// TIA Portal V19 export
FUNCTION "@CmMotor" : Void   // FC2004, STL
TITLE = Control Module for Motor/Pump - Fixed Speed
{ S7_Optimized_Access := 'FALSE' }
AUTHOR : FoodSystem(AlfaLaval)
FAMILY : ControlModule
NAME : CM005
VERSION : 3.5
// Date        Rev      Change                                           Changed by
// ---------------------------------------------------------------------------------------------------------------------------------
// 08.04.2022 V3.0       Update                                    Food System (Alfalaval)
// 
// 28.07.2022 V3.1       Update                                    Food System (Alfalaval)
// 
// 14.11.2022 V3.2       Update                                    Food System (Alfalaval)
// 
// 26.12.2022 V3.3       Update                                    Food System (Alfalaval)
// 
// 16.05.2023 V3.4       Update                                    Food System (Alfalaval)
// 
// 01.12.2023 V3.5       Update                                    Food System (Alfalaval)
// ---------------------------------------------------------------------------------------------------------------------------------
// Motor with 3 Inputs and 1 output
// 1. Running Feedback, 2. Tripped Feedback, 3. Remote Feedback
// and 1. Start O/P
// The CM_Motor controls and monitors a single-speed one direction motor. 
// Additionally it also supports functions like feedback monitoring and alarm 
// generation, simulation and displays status to the HMI
// Date        Rev      Change                                           Changed by
// ---------------------------------------------------------------------------------------------------------------------------------
// 08.04.2022 V3.0       Update                                    Food System (Alfalaval)
// 
// 28.07.2022 V3.1       Update                                    Food System (Alfalaval)
// 
// 14.11.2022 V3.2       Update                                    Food System (Alfalaval)
// ---------------------------------------------------------------------------------------------------------------------------------
// Motor with 3 Inputs and 1 output
// 1. Running Feedback, 2. Tripped Feedback, 3. Remote Feedback
// and 1. Start O/P
// The CM_Motor controls and monitors a single-speed one direction motor. 
// Additionally it also supports functions like feedback monitoring and alarm 
// generation, simulation and displays status to the HMI
// stored: AutoNumber false
   VAR_INPUT
      i_Remote : Bool;   // Local / Remote
      i_RunFb : Bool;   // Motor Run Feedback
      i_TrippedFb : Bool;   // Motor Tripped Feedback
      i_Inhibit : Bool;   // 0 = Interlock, 1 = Healthy. Motor Inhibit
      i_EStop : Bool;   // Emergency Stop
      FeatureITripPolarity : Bool;   // Set 0 (I_TrippedFb --> 0 = Tripped), Set 1 (I_TrippedFb --> 1 = Tripped) Only for Trip HW Signal.
      FirstScanBit : Bool;   // First Scan Bit
      OneSec : Bool;   // One Second Pulse
      SimOn : Bool;   // Activate Simulation
      SimOff : Bool;   // Deactivate Simulation
      CommonReset : Bool;   // Reset fault
      HooterReset : Bool;   // Reset Hooter
      AutoReqMode : Bool;   // Activate PLC Auto Mode
      DCSOperation : Bool;   // Request from DCS to operate command from DCS
   END_VAR
   VAR_OUTPUT
      q_On : Bool;   // Motor run output
   END_VAR
   VAR_IN_OUT
      CM : Any;   // Parameter for control module
   END_VAR
   VAR_TEMP
      UDTMotor : "UDT CM_Motor";   // UDT data for for control module
      Pointer : DWord;   // Pointer for storage UDT
      DB : Word;   // UDT DB for data load
      TempQAutoOn : Bool;   // Internal on command in Auto mode before start interlock
      TempQManON : Bool;   // Internal on command in manual mode
      Permissive : Struct   // Temp Bits for Start Interlock Processing
         Inlk0 : Bool;
         Inlk1 : Bool;
         Inlk2 : Bool;
         Inlk3 : Bool;
         Inlk4 : Bool;
         Inlk5 : Bool;
         Inlk6 : Bool;
         Inlk7 : Bool;
         Inlk8 : Bool;
         Inlk9 : Bool;
         Inlk10 : Bool;
         Inlk11 : Bool;
         Inlk12 : Bool;
         Inlk13 : Bool;
         Inlk14 : Bool;
         Inlk15 : Bool;
      END_STRUCT;
      Interlock : Struct   // Temp Bits for Run Interlock Processing
         Inlk0 : Bool;
         Inlk1 : Bool;
         Inlk2 : Bool;
         Inlk3 : Bool;
         Inlk4 : Bool;
         Inlk5 : Bool;
         Inlk6 : Bool;
         Inlk7 : Bool;
         Inlk8 : Bool;
         Inlk9 : Bool;
         Inlk10 : Bool;
         Inlk11 : Bool;
         Inlk12 : Bool;
         Inlk13 : Bool;
         Inlk14 : Bool;
         Inlk15 : Bool;
      END_STRUCT;
      BypassPermissive : Struct   // Temp Bits for Bypass Start Interlock Processing
         Inlk0 : Bool;
         Inlk1 : Bool;
         Inlk2 : Bool;
         Inlk3 : Bool;
         Inlk4 : Bool;
         Inlk5 : Bool;
         Inlk6 : Bool;
         Inlk7 : Bool;
         Inlk8 : Bool;
         Inlk9 : Bool;
         Inlk10 : Bool;
         Inlk11 : Bool;
         Inlk12 : Bool;
         Inlk13 : Bool;
         Inlk14 : Bool;
         Inlk15 : Bool;
      END_STRUCT;
      BypassInterlock : Struct   // Temp Bits for Bypass Run Interlock Processing
         Inlk0 : Bool;
         Inlk1 : Bool;
         Inlk2 : Bool;
         Inlk3 : Bool;
         Inlk4 : Bool;
         Inlk5 : Bool;
         Inlk6 : Bool;
         Inlk7 : Bool;
         Inlk8 : Bool;
         Inlk9 : Bool;
         Inlk10 : Bool;
         Inlk11 : Bool;
         Inlk12 : Bool;
         Inlk13 : Bool;
         Inlk14 : Bool;
         Inlk15 : Bool;
      END_STRUCT;
   END_VAR
BEGIN

NETWORK
TITLE = LOAD DATA FROM DB

      L     P##CM;  // Any datapointer for CM
      LAR1;
      L     W [AR1, P#4.0];
      T     #DB;  // Number of DB
      L     D [AR1, P#6.0];
      T     #Pointer;  // Pointer for data
      LAR1;

      OPN   DB [#DB];
      L     W [AR1, P#0.0];  // Data transfer to Local Area
      T     %LW0;

      L     W [AR1, P#2.0];  // Data transfer to Local Area
      T     %LW2;


      L     W [AR1, P#4.0];  // Data transfer to Local Area
      T     %LW4;

      L     W [AR1, P#6.0];  // Data transfer to Local Area
      T     %LW6;


      L     W [AR1, P#8.0];  // Data transfer to Local Area
      T     #UDTMotor.FTRSet;

      L     W [AR1, P#10.0];  // Data transfer to Local Area
      T     #UDTMotor.FTSSet;

      L     W [AR1, P#12.0];  // Data transfer to Local Area
      T     #UDTMotor.FTRActual;

      L     W [AR1, P#14.0];  // Data transfer to Local Area
      T     #UDTMotor.FTSActual;

      L     W [AR1, P#16.0];  // Data transfer to Local Area
      T     #UDTMotor.ARH;

      L     W [AR1, P#18.0];  // Data transfer to Local Area
      T     #UDTMotor.Display;

      L     W [AR1, P#20.0];  // Data transfer to Local Area
      T     #UDTMotor.TempARH;


      L     W [AR1, P#22.0];  // Data transfer to Local Area
      T     #UDTMotor.PulseTimeStart;

      L     W [AR1, P#24.0];  // Data transfer to Local Area
      T     #UDTMotor.PulseTimeStop;

      L     W [AR1, P#26.0];  // Data transfer to Local Area
      T     #UDTMotor.BypassPermissive;

      L     W [AR1, P#28.0];  // Data transfer to Local Area
      T     #UDTMotor.BypassInterlock;

      L     W [AR1, P#30.0];  // Data transfer to Local Area
      T     %LW30;

      L     W [AR1, P#32.0];  // Data transfer to Local Area
      T     %LW32;

      L     W [AR1, P#34.0];  // Data transfer to Local Area
      T     #UDTMotor.AlarmHmi;

      L     W [AR1, P#36.0];  // Data transfer to Local Area
      T     #UDTMotor.ActiveTime;


      L     W [AR1, P#38.0];  // Data transfer to Local Area
      T     #UDTMotor.MotorType;

      L     D [AR1, P#40.0];  // Data transfer to Local Area
      T     #UDTMotor.Spare2;

      L     D [AR1, P#44.0];  // Data transfer to Local Area
      T     %LD44;  // oBJECT enable

      L     W [AR1, P#48.0];  // Data transfer to Local Area
      T     %LW48;  // FP EDGES


NETWORK
TITLE = RESET MANUAL COMMAND AND RESET ALARMS BY FIRST_SCAN_BIT
// On Power on and Off Motor start commond should reset.
      A     #FirstScanBit;  // First Scan
      R     #UDTMotor.Command.ManRun;  // Manual Start Commonad
      R     #UDTMotor.Status.FTR;  // Motor/Pump Fail to Run Fault.(FTR)
      R     #UDTMotor.Status.FTS;  // Motor/Pump Fail to Stop Fault.(FTS)


NETWORK
TITLE = Operation from DCS=1 (Disable command buttons from HMI)
      A     #DCSOperation;
      ON    #i_Remote;
      =     #UDTMotor.Command.DCSOperation;
      =     #UDTMotor.ObjEn.AlarmMask;
      =     #UDTMotor.ObjEn.Auto;
      =     #UDTMotor.ObjEn.Manual;
      =     #UDTMotor.ObjEn.ByInlk;
      =     #UDTMotor.ObjEn.ByPer;
      =     #UDTMotor.ObjEn.FTRSetpointEn;
      =     #UDTMotor.ObjEn.FTSSetpointEn;
      =     #UDTMotor.ObjEn.Reset;
      =     #UDTMotor.ObjEn.SimOn;
      =     #UDTMotor.ObjEn.ResetARH;

      A     #DCSOperation;
      ON    #i_Remote;
      O     #UDTMotor.Status.Mode;
      =     #UDTMotor.ObjEn.Start;


NETWORK
TITLE = LOAD INTERLOCK TO TEMP
// ----------------------------------------------------------------------------------------------//
//                                  READ INTERLOCK STATUS TO TEMP                                 //
// ----------------------------------------------------------------------------------------------//
      L     %LW30;  // Load start intrlocks
      T     %LW62;  // Save into TEMP
      L     %LW32;  // Load run intrlocks
      T     %LW64;  // Save into TEMP
      L     #UDTMotor.BypassPermissive;  // Load bypass start intrlocks
      T     %LW66;  // Save into TEMP
      L     #UDTMotor.BypassInterlock;  // Load bypass run intrlocks
      T     %LW68;  // Save into TEMP


NETWORK
TITLE = Reset Start Permissive & Run Interlock Bypasses
      A     #UDTMotor.Command.ResetRunPermissiveILByp;  // Check if Reset Interlock Bypass Bit is True

      JCN   INTBYPS_RST;  // Jump if the Reset Interlock Bypass bit is False

      L     16#0;
      T     #UDTMotor.BypassInterlock;  // Transfer 0 to Temp  Interlock Bypass permissive bits
      T     %LW68;  // Transfer 0 to Temp Interlock Bypass bits

INTBYPS_RST:NOP   0;


      A     #UDTMotor.Command.ResetStartPermissiveILByp;  // Check if Reset Permissive Bypass Bit is True

      JCN   PERBYPS_RST;  // Jump if the Reset Permissive Bypass bit is False

      L     16#0;  // Load 0
      T     #UDTMotor.BypassPermissive;  // Transfer 0 to Temp Permissive Bypass permissive bits
      T     %LW66;  // Transfer 0 to Temp Permissive Bypass bits

PERBYPS_RST:NOP   0;

NETWORK
TITLE = START INTERLOCK LOGIC
// ----------------------------------------------------------------------------------------------//
//                              OVERWRITE BYPASS BIT DUE TO NAMEPLATE                            //
// ----------------------------------------------------------------------------------------------//
//       CLR
//       =     #BypassPermissive.Inlk8// If bypass8
//       =     #BypassPermissive.Inlk9// If bypass9
//       =     #BypassPermissive.Inlk10// If bypass10
//       =     #BypassPermissive.Inlk11// If bypass11
//       =     #BypassPermissive.Inlk12// If bypass12
//       =     #BypassPermissive.Inlk13// If bypass13
//       =     #BypassPermissive.Inlk14// If bypass14
//       =     #BypassPermissive.Inlk15// If bypass15
//       SET
//       =     #Permissive.Inlk8    // Interlock8
//       =     #Permissive.Inlk9    // Interlock9
//       =     #Permissive.Inlk10   // Interlock10
//       =     #Permissive.Inlk11   // Interlock11
//       =     #Permissive.Inlk12   // Interlock12
//       =     #Permissive.Inlk13   // Interlock13
//       =     #Permissive.Inlk14   // Interlock14
//       =     #Permissive.Inlk15   // Interlock15



//----------------------------------------------------------------------------------------------//
//                                      START INTERLOCK LOGIC                                   //
//----------------------------------------------------------------------------------------------//

      A     #BypassPermissive.Inlk0;  // If bypass0
      JC    START;
      AN    #Permissive.Inlk0;  // If interlock
      JCN   START;
      R     #UDTMotor.Status.Permissive;  //RESET OK INTERLOCKS
      JU    ST_INT;  // out
START:NOP   0;

      A     #BypassPermissive.Inlk1;  // If bypass1
      JC    START1;
      AN    #Permissive.Inlk1;  // If interlock1
      JCN   START1;
      R     #UDTMotor.Status.Permissive;  //RESET OK INTERLOCKS
      JU    ST_INT;  // out
START1:NOP   0;

      A     #BypassPermissive.Inlk2;  // If bypass2
      JC    START2;
      AN    #Permissive.Inlk2;  // If interlock2
      JCN   START2;
      R     #UDTMotor.Status.Permissive;  //RESET OK INTERLOCKS
      JU    ST_INT;  // out
START2:NOP   0;

      A     #BypassPermissive.Inlk3;  // If bypass3
      JC    START3;
      AN    #Permissive.Inlk3;  // If interlock3
      JCN   START3;
      R     #UDTMotor.Status.Permissive;  //RESET OK INTERLOCKS
      JU    ST_INT;  // out
START3:NOP   0;

      A     #BypassPermissive.Inlk4;  // If bypass4
      JC    START4;
      AN    #Permissive.Inlk4;  // If interlock4
      JCN   START4;
      R     #UDTMotor.Status.Permissive;  //RESET OK INTERLOCKS
      JU    ST_INT;  // out
START4:NOP   0;

      A     #BypassPermissive.Inlk5;  // If bypass5
      JC    START5;
      AN    #Permissive.Inlk5;  // If interlock5
      JCN   START5;
      R     #UDTMotor.Status.Permissive;  //RESET OK INTERLOCKS
      JU    ST_INT;  // out
START5:NOP   0;

      A     #BypassPermissive.Inlk6;  // If bypass6
      JC    START6;
      AN    #Permissive.Inlk6;  // If interlock6
      JCN   START6;
      R     #UDTMotor.Status.Permissive;  //RESET OK INTERLOCKS
      JU    ST_INT;  // out
START6:NOP   0;

      A     #BypassPermissive.Inlk7;  // If bypass7
      JC    START7;
      AN    #Permissive.Inlk7;  // If interlock7
      JCN   START7;
      R     #UDTMotor.Status.Permissive;  //RESET OK INTERLOCKS
      JU    ST_INT;  // out
START7:NOP   0;

      A     #BypassPermissive.Inlk8;  // If bypass8
      JC    START8;
      AN    #Permissive.Inlk8;  // If interlock8
      JCN   START8;
      R     #UDTMotor.Status.Permissive;  //RESET OK INTERLOCKS
      JU    ST_INT;  // out
START8:NOP   0;

      A     #BypassPermissive.Inlk9;  // If bypass9
      JC    START9;
      AN    #Permissive.Inlk9;  // If interlock9
      JCN   START9;
      R     #UDTMotor.Status.Permissive;  //RESET OK INTERLOCKS
      JU    ST_INT;  // out
START9:NOP   0;

      A     #BypassPermissive.Inlk10;  // If bypass10
      JC    START10;
      AN    #Permissive.Inlk10;  // If interlock10
      JCN   START10;
      R     #UDTMotor.Status.Permissive;  //RESET OK INTERLOCKS
      JU    ST_INT;  // out
START10:NOP   0;

      A     #BypassPermissive.Inlk11;  // If bypass11
      JC    START11;
      AN    #Permissive.Inlk11;  // If interlock11
      JCN   START11;
      R     #UDTMotor.Status.Permissive;  //RESET OK INTERLOCKS
      JU    ST_INT;  // out
START11:NOP   0;

      A     #BypassPermissive.Inlk12;  // If bypass12
      JC    START12;
      AN    #Permissive.Inlk12;  // If interlock12
      JCN   START12;
      R     #UDTMotor.Status.Permissive;  //RESET OK INTERLOCKS
      JU    ST_INT;  // out
START12:NOP   0;

      A     #BypassPermissive.Inlk13;  // If bypass13
      JC    START13;
      AN    #Permissive.Inlk13;  // If interlock13
      JCN   START13;
      R     #UDTMotor.Status.Permissive;  //RESET OK INTERLOCKS
      JU    ST_INT;  // out
START13:NOP   0;

      A     #BypassPermissive.Inlk14;  // If bypass14
      JC    START14;
      AN    #Permissive.Inlk14;  // If interlock14
      JCN   START14;
      R     #UDTMotor.Status.Permissive;  //RESET OK INTERLOCKS
      JU    ST_INT;  // out
START14:NOP   0;

      A     #BypassPermissive.Inlk15;  // If bypass15
      JC    START15;
      AN    #Permissive.Inlk15;  // If interlock15
      JCN   START15;
      R     #UDTMotor.Status.Permissive;  //RESET OK INTERLOCKS
      JU    ST_INT;  // out
START15:NOP   0;

      SET;
      =     #UDTMotor.Status.Permissive;  //SET OK INTERLOCKS
ST_INT:NOP   0;

NETWORK
TITLE = RUN INTERLOCK LOGIC
// ----------------------------------------------------------------------------------------------//
//                              OVERWRITE BYPASS BIT DUE TO NAMEPLATE                            //
// ----------------------------------------------------------------------------------------------//
//       CLR
//       =     #BypassInterlock.Inlk8// If bypass8
//       =     #BypassInterlock.Inlk9// If bypass9
//       =     #BypassInterlock.Inlk10// If bypass10
//       =     #BypassInterlock.Inlk11// If bypass11
//       =     #BypassInterlock.Inlk12// If bypass12
//       =     #BypassInterlock.Inlk13// If bypass13
//       =     #BypassInterlock.Inlk14// If bypass14
//       =     #BypassInterlock.Inlk15// If bypass15
//       SET
//       =     #Interlock.Inlk8     // Interlock8
//       =     #Interlock.Inlk9     // Interlock9
//       =     #Interlock.Inlk10    // Interlock10
//       =     #Interlock.Inlk11    // Interlock11
//       =     #Interlock.Inlk12    // Interlock12
//       =     #Interlock.Inlk13    // Interlock13
//       =     #Interlock.Inlk14    // Interlock14
//       =     #Interlock.Inlk15    // Interlock15


//----------------------------------------------------------------------------------------------//
//                                        RUN INTERLOCK LOGIC                                   //
//----------------------------------------------------------------------------------------------//
      A     #BypassInterlock.Inlk0;  // If bypass
      JC    RUN;
      AN    #Interlock.Inlk0;  // If interlock
      JCN   RUN;
      R     #UDTMotor.Status.Interlock;  //RESET OK INTERLOCKS
      JU    RUN_INT;  // out
RUN:  NOP   0;

      A     #BypassInterlock.Inlk1;  // If bypass1
      JC    RUN1;
      AN    #Interlock.Inlk1;  // If interlock1
      JCN   RUN1;
      R     #UDTMotor.Status.Interlock;  //RESET OK INTERLOCKS
      JU    RUN_INT;  // out
RUN1: NOP   0;

      A     #BypassInterlock.Inlk2;  // If bypass2
      JC    RUN2;
      AN    #Interlock.Inlk2;  // If interlock2
      JCN   RUN2;
      R     #UDTMotor.Status.Interlock;  //RESET OK INTERLOCKS
      JU    RUN_INT;  // out
RUN2: NOP   0;

      A     #BypassInterlock.Inlk3;  // If bypass3
      JC    RUN3;
      AN    #Interlock.Inlk3;  // If interlock3
      JCN   RUN3;
      R     #UDTMotor.Status.Interlock;  //RESET OK INTERLOCKS
      JU    RUN_INT;  // out
RUN3: NOP   0;

      A     #BypassInterlock.Inlk4;  // If bypass4
      JC    RUN4;
      AN    #Interlock.Inlk4;  // If interlock4
      JCN   RUN4;
      R     #UDTMotor.Status.Interlock;
      JU    RUN_INT;
RUN4: NOP   0;

      A     #BypassInterlock.Inlk5;  // If bypass5
      JC    RUN5;
      AN    #Interlock.Inlk5;  // If interlock5
      JCN   RUN5;
      R     #UDTMotor.Status.Interlock;  //RESET OK INTERLOCKS
      JU    RUN_INT;  // out
RUN5: NOP   0;

      A     #BypassInterlock.Inlk6;  // If bypass6
      JC    RUN6;
      AN    #Interlock.Inlk6;  // If interlock6
      JCN   RUN6;
      R     #UDTMotor.Status.Interlock;  //RESET OK INTERLOCKS
      JU    RUN_INT;  // out
RUN6: NOP   0;

      A     #BypassInterlock.Inlk7;  // If bypass7
      JC    RUN7;
      AN    #Interlock.Inlk7;  // If interlock7
      JCN   RUN7;
      R     #UDTMotor.Status.Interlock;  //RESET OK INTERLOCKS
      JU    RUN_INT;  // out
RUN7: NOP   0;

      A     #BypassInterlock.Inlk8;  // If bypass8
      JC    RUN8;
      AN    #Interlock.Inlk8;  // If interlock8
      JCN   RUN8;
      R     #UDTMotor.Status.Interlock;  //RESET OK INTERLOCKS
      JU    RUN_INT;  // out
RUN8: NOP   0;

      A     #BypassInterlock.Inlk9;  // If bypass9
      JC    RUN9;
      AN    #Interlock.Inlk9;  // If interlock9
      JCN   RUN9;
      R     #UDTMotor.Status.Interlock;  //RESET OK INTERLOCKS
      JU    RUN_INT;  // out
RUN9: NOP   0;

      A     #BypassInterlock.Inlk10;  // If bypass10
      JC    RUN10;
      AN    #Interlock.Inlk10;  // If interlock10
      JCN   RUN10;
      R     #UDTMotor.Status.Interlock;  //RESET OK INTERLOCKS
      JU    RUN_INT;  // out
RUN10:NOP   0;

      A     #BypassInterlock.Inlk11;  // If bypass11
      JC    RUN11;
      AN    #Interlock.Inlk11;  // If interlock11
      JCN   RUN11;
      R     #UDTMotor.Status.Interlock;  //RESET OK INTERLOCKS
      JU    RUN_INT;  // out
RUN11:NOP   0;

      A     #BypassInterlock.Inlk12;  // If bypass12
      JC    RUN12;
      AN    #Interlock.Inlk12;  // If interlock12
      JCN   RUN12;
      R     #UDTMotor.Status.Interlock;  //RESET OK INTERLOCKS
      JU    RUN_INT;  // out
RUN12:NOP   0;

      A     #BypassInterlock.Inlk13;  // If bypass13
      JC    RUN13;
      AN    #Interlock.Inlk13;  // If interlock13
      JCN   RUN13;
      R     #UDTMotor.Status.Interlock;  //RESET OK INTERLOCKS
      JU    RUN_INT;  // out
RUN13:NOP   0;

      A     #BypassInterlock.Inlk14;  // If bypass14
      JC    RUN14;
      AN    #Interlock.Inlk14;  // If interlock14
      JCN   RUN14;
      R     #UDTMotor.Status.Interlock;  //RESET OK INTERLOCKS
      JU    RUN_INT;  // out
RUN14:NOP   0;

      A     #BypassInterlock.Inlk15;  // If bypass15
      JC    RUN15;
      AN    #Interlock.Inlk15;  // If interlock15
      JCN   RUN15;
      R     #UDTMotor.Status.Interlock;  //RESET OK INTERLOCKS
      JU    RUN_INT;  // out
RUN15:NOP   0;


      SET;
      =     #UDTMotor.Status.Interlock;  //SET OK INTERLOCKS
RUN_INT:NOP   0;


NETWORK
TITLE = SIMULATION MODE / SIMULATIONSMODUS

//----------------------------------------------------------------------------------------------//
//                             Simulation order from HMI/SCADA                                  //
//----------------------------------------------------------------------------------------------//
      A     #SimOn;  // Request simulation ON from HMI/SCADA
      FP    #UDTMotor.FP.SimOn;  //Front positive pulse
      S     #UDTMotor.Command.SimOn;  //Simulation ON command from current nameplate
      R     #UDTMotor.Command.SimOff;  //Simulation OFF command from current nameplate

      A     #UDTMotor.Command.SimOn;  //Simulation ON command from current nameplate
      S     #UDTMotor.Status.SimOn;  //Simulation ON status
      R     #UDTMotor.Status.SimOff;  //Simulation OFF status

      A     #SimOff;  // Request simulation OFF from HMI/SCADA
      FP    #UDTMotor.FP.SimOff;  //Front positive pulse
      S     #UDTMotor.Command.SimOff;  //Simulation OFF command from current nameplate
      R     #UDTMotor.Command.SimOn;  //Simulation ON command from current nameplate

      A     #UDTMotor.Command.SimOff;  //Simulation OFF command from current nameplate
      S     #UDTMotor.Status.SimOff;  //Simulation OFF status
      R     #UDTMotor.Status.SimOn;  //Simulation ON status
//----------------------------------------------------------------------------------------------//
//                    If no one simulation command present - initialisation PLC                 //
//----------------------------------------------------------------------------------------------//
      AN    #UDTMotor.Command.SimOn;  //Simulation ON command from current nameplate
      AN    #UDTMotor.Command.SimOff;  //Simulation OFF command from current nameplate
      S     #UDTMotor.Command.SimOff;  //Simulation OFF command from current nameplate
//----------------------------------------------------------------------------------------------//
//                             Simulation order from current nameplate                          //
//----------------------------------------------------------------------------------------------//
      A     #UDTMotor.Command.SimOn;  //Simulation ON command from current nameplate
      FP    #UDTMotor.FP.SimulationOn;  //Front positive pulse
      R     #UDTMotor.Command.SimOff;  //Simulation OFF command from current nameplate

      A     #UDTMotor.Command.SimOff;  //Simulation OFF command from current nameplate
      FP    #UDTMotor.FP.SimulationOff;  //Front positive pulse
      R     #UDTMotor.Command.SimOn;  //Simulation ON command from current nameplate



NETWORK
TITLE = STATUS MAPPING
// ----------------------------------------------------------------------------------------------//
//                                   MAPPING SIGNAL FOR HMI/SCADA                                //
// ----------------------------------------------------------------------------------------------//


      A     #UDTMotor.Status.Permissive;  //START OK INTERLOCKS
      A     #UDTMotor.Status.Interlock;  //RUN OK INTERLOCKS
      =     #UDTMotor.Status.Interlocked;  //STATUS OK INTERLOCKS

      A     #i_EStop;  //ESTOP RELAY
      =     #UDTMotor.Status.Estop;  // STATUS ESTOP OK

      A     #UDTMotor.Command.AutoRun;  // AUTO ACTION REQUEST
      =     #UDTMotor.Status.AutoActionRequest;  // STATUS AUTO ACTION REQUEST

      A     #i_Remote;  // Motor/Pump in remote mode
      =     #UDTMotor.Status.Remote;  // Motor/Pump in remote mode

      A     #i_Inhibit;
      =     #UDTMotor.Status.Inhibit;


      A     #UDTMotor.Command.ManRun;  // MANUAL ACTION REQUEST
      =     #UDTMotor.Status.ManualActionRequest;  // STATUS MANUAL ACTION REQUEST

      A     #UDTMotor.Command.AlarmMask;  // ALARM MASK REQUEST
      =     #UDTMotor.Status.AlarmMask;  // STATUS ALARM MASK


// |************************************************************************|
// |                     Feedback Simulation logic                          |
// |************************************************************************|

      AN    #UDTMotor.Command.SimOn;  // Motor/Pump Run Feedback Simulatione
      A     #i_RunFb;  // Motor/Pump Run Feedback from field
      O;
      A     #UDTMotor.Command.SimOn;  // Motor/Pump Run Feedback Simulatione
      A     #UDTMotor.Status.QOn;  // Motor/Pump internal output
      =     #UDTMotor.Status.RunFb;  // Motor/Pump Running feedback for SCADA and FTR logic


// |************************************************************************|
// |                     Process signal mapping to HMI                         |
// |************************************************************************|

      A     #UDTMotor.Command.Mode;
      =     #UDTMotor.Status.Mode;


// Local and Auto/Man Display on HMI [ICON] on Priority

      AN    #UDTMotor.Status.Remote;
      A(;
      ON    #UDTMotor.Status.Mode;
      O     #UDTMotor.Status.Mode;
      );
      =     #UDTMotor.Status.LocalRemoteIcon;

// Manual Mode Display On HMI [ICON]

      AN    #UDTMotor.Status.Mode;
      A     #UDTMotor.Status.Remote;
      AN    #UDTMotor.Status.LocalRemoteIcon;
      =     #UDTMotor.Status.AMStatusIcon;


//----------------------------------------------------------------------------------------------//
//                               ABNORMAL_ICON                                                  //
//----------------------------------------------------------------------------------------------//
      A     #UDTMotor.Command.AlarmMask;  // Fault are masked
      ON    #UDTMotor.Status.Interlocked;  //STATUS OK INTERLOCKS
      O     #UDTMotor.Status.InlkBypassIcon;
      ON    #UDTMotor.Status.InlkStatusIcon;  //HMI sign
      ON    #i_EStop;
      O     #UDTMotor.Status.SimOn;  //Simulation ON command from current nameplate
      =     #UDTMotor.Status.AbnormalIcon;  // Abnormal icon on HMI/SCADA


//----------------------------------------------------------------------------------------------//
//                                  BYPASS INTERLOCK FOR HMI/SCADA                              //
//----------------------------------------------------------------------------------------------//
      CLR;
      A     #BypassPermissive.Inlk0;  // If bypass
      O     #BypassPermissive.Inlk1;  // If bypass1
      O     #BypassPermissive.Inlk2;  // If bypass2
      O     #BypassPermissive.Inlk3;  // If bypass3
      O     #BypassPermissive.Inlk4;  // If bypass4
      O     #BypassPermissive.Inlk5;  // If bypass5
      O     #BypassPermissive.Inlk6;  // If bypass6
      O     #BypassPermissive.Inlk7;  // If bypass7
      O     #BypassPermissive.Inlk8;  // If bypass8
      O     #BypassPermissive.Inlk9;  // If bypass9
      O     #BypassPermissive.Inlk10;  // If bypass10
      O     #BypassPermissive.Inlk11;  // If bypass11
      O     #BypassPermissive.Inlk12;  // If bypass12
      O     #BypassPermissive.Inlk13;  // If bypass13
      O     #BypassPermissive.Inlk14;  // If bypass14
      O     #BypassPermissive.Inlk15;  // If bypass15

      O     #BypassInterlock.Inlk0;  // If bypass
      O     #BypassInterlock.Inlk1;  // If bypass1
      O     #BypassInterlock.Inlk2;  // If bypass2
      O     #BypassInterlock.Inlk3;  // If bypass3
      O     #BypassInterlock.Inlk4;  // If bypass4
      O     #BypassInterlock.Inlk5;  // If bypass5
      O     #BypassInterlock.Inlk6;  // If bypass6
      O     #BypassInterlock.Inlk7;  // If bypass7
      O     #BypassInterlock.Inlk8;  // If bypass8
      O     #BypassInterlock.Inlk9;  // If bypass9
      O     #BypassInterlock.Inlk10;  // If bypass10
      O     #BypassInterlock.Inlk11;  // If bypass11
      O     #BypassInterlock.Inlk12;  // If bypass12
      O     #BypassInterlock.Inlk13;  // If bypass13
      O     #BypassInterlock.Inlk14;  // If bypass14
      O     #BypassInterlock.Inlk15;  // If bypass15
      =     #UDTMotor.Status.InlkBypassIcon;
//----------------------------------------------------------------------------------------------//
//                                         INTERLOCK FOR HMI/SCADA                              //
//----------------------------------------------------------------------------------------------//

      A     #UDTMotor.Status.QOn;  // If Motor internal run command True.
      JC    BYPS_PERM_0;  // Jump to Run Interlock do not check Permissives

      A     #Permissive.Inlk0;  // Interlock
      A     #Permissive.Inlk1;  // Interlock1
      A     #Permissive.Inlk2;  // Interlock2
      A     #Permissive.Inlk3;  // Interlock3
      A     #Permissive.Inlk4;  // Interlock4
      A     #Permissive.Inlk5;  // Interlock5
      A     #Permissive.Inlk6;  // Interlock6
      A     #Permissive.Inlk7;  // Interlock7
      A     #Permissive.Inlk8;  // Interlock8
      A     #Permissive.Inlk9;  // Interlock9
      A     #Permissive.Inlk10;  // Interlock10
      A     #Permissive.Inlk11;  // Interlock11
      A     #Permissive.Inlk12;  // Interlock12
      A     #Permissive.Inlk13;  // Interlock13
      A     #Permissive.Inlk14;  // Interlock14
      A     #Permissive.Inlk15;  // Interlock15
BYPS_PERM_0:NOP   0;
      A     #Interlock.Inlk0;  // Interlock
      A     #Interlock.Inlk1;  // Interlock1
      A     #Interlock.Inlk2;  // Interlock2
      A     #Interlock.Inlk3;  // Interlock3
      A     #Interlock.Inlk4;  // Interlock4
      A     #Interlock.Inlk5;  // Interlock5
      A     #Interlock.Inlk6;  // Interlock6
      A     #Interlock.Inlk7;  // Interlock7
      A     #Interlock.Inlk8;  // Interlock8
      A     #Interlock.Inlk9;  // Interlock9
      A     #Interlock.Inlk10;  // Interlock10
      A     #Interlock.Inlk11;  // Interlock11
      A     #Interlock.Inlk12;  // Interlock12
      A     #Interlock.Inlk13;  // Interlock13
      A     #Interlock.Inlk14;  // Interlock14
      A     #Interlock.Inlk15;  // Interlock15
      =     #UDTMotor.Status.InlkStatusIcon;  //HMI sign



NETWORK
TITLE = MANUAL COMMAND/MODE LOGIC
// Motor/Pump Ready to start Condition derived from following bits: -
// 
// a) Auto = Logic 1.
// b) Available = Logic 1
// c) No Fault
// d) Start Interlock and Process Intelock Healthy
// |************************************************************************|
// |                           RTS Display Logic                            |
// |************************************************************************|
      A     #UDTMotor.Status.Remote;  // Motor/Pump in remote mode
      AN    #UDTMotor.Status.Tripped;  // Motor/Pump tripped
      AN    #UDTMotor.Status.QOn;  // Start Command not Present
      AN    #UDTMotor.Status.GeneralFault;  // Motor/Pump Healthy
      A     #UDTMotor.Status.Permissive;  // Motor/Pump Start interlock in heatly condition
      A     #UDTMotor.Status.Interlock;  // Motor/Pump Process interlock in heatly condition
      A     #i_Inhibit;  // Motor/Pump inhitbit
      =     #UDTMotor.Status.RTS;  // Motor/Pump Ready to start (RTS BIT for dispaly on HMI)



// |************************************************************************|
// |    Maintaining Same state From PLC Auto to PLC Manual Transfer         |
// |************************************************************************|

      A     #UDTMotor.Status.QOn;  // Start Command Present
      ON    #UDTMotor.Status.Interlocked;  // INTERLOCK PRESENT
      A(;  // AND
      AN    #UDTMotor.Status.Mode;  // Motor/Pump selected in PLC Manual Mode
      FP    #UDTMotor.Command.FP1;  // Change detected
      );  // yes! Then
      S     #UDTMotor.Command.ManRun;  // Set Motor/Pump Start command from the HMI



// |************************************************************************|
// |                      PLC Auto Start-Stop Logic                         |
// |************************************************************************|

      A     #AutoReqMode;
      O     #UDTMotor.Command.AutoModeReq;
      FP    #UDTMotor.FP.AutoReq;
      S     #UDTMotor.Command.Mode;  // Auto MODE



// |************************************************************************|
// |                      PLC Manual Start-Stop Logic                       |
// |************************************************************************|

      A     #UDTMotor.Status.Remote;  // Motor/Pump in remote mode
      AN    #UDTMotor.Status.Tripped;  // Motor/Pump tripped
      AN    #UDTMotor.Status.GeneralFault;  // Motor/Pump Healthy Signal is Logic 1
      AN    #UDTMotor.Status.Mode;  // Motor/Pump PLC Manual selected from HMI
      A     #UDTMotor.Command.ManRun;  // Motor/Pump Start - Stop command from HMI
      A     #UDTMotor.Status.Interlock;  // Motor/Pump Process Interlock are healthy
      A     #i_Inhibit;  // Motor/Pump inhitbit
      A     #i_EStop;
      =     #TempQManON;  // Internal on command in manual mode



// |************************************************************************|
// |                      PLC Auto Start-Stop Logic                         |
// |************************************************************************|

      A     #UDTMotor.Status.Remote;  // Motor/Pump in remote mode
      AN    #UDTMotor.Status.Tripped;  // Motor/Pump tripped
      AN    #UDTMotor.Status.GeneralFault;  // Motor/Pump Healthy Signal is Logic 1
      A     #UDTMotor.Status.Mode;  // Motor/Pump PLC Auto selected from the HMI
      A     #UDTMotor.Command.AutoRun;  // Motor/Pump Auto Run Switch interlock healthy
      A     #UDTMotor.Status.Interlock;  // Motor/Pump Process Interlock are healthy
      A     #i_Inhibit;  // Motor/Pump inhitbit
      A     #i_EStop;
      =     #TempQAutoOn;  // Internal on command in Auto mode before start interlock



// |************************************************************************|
// |                              Auto / Manual conditions                  |
// |************************************************************************|

      A(;
      O     #TempQAutoOn;  // Internal on command before start interlock
      O     #TempQManON;  // Internal on command in manual mode
      );
      A(;
      O     #UDTMotor.Status.Permissive;  // Motor/Pump Start Interlock are healthy
      O     #UDTMotor.Status.QOn;  // Motor/Pump Start Command Flag in PLC Auto Mode
      );
      =     #UDTMotor.Status.QOn;  // Motor/Pump Start Command Flag



// |************************************************************************|
// |                     Deactivate Manual Start Command                    |
// |************************************************************************|


      ON    #UDTMotor.Status.Remote;  // Motor/Pump in local mode
      O     #UDTMotor.Status.GeneralFault;  // Motor/Pump Healthy Signal is Logic 0
      O     #UDTMotor.Status.DiscrFault;  // Motor Discrepancy
      ON    #i_Inhibit;  // Motor/Pump inhitbit
      ON    #UDTMotor.Status.QOn;  // Motor/Pump Start Command Flag
      ON    #i_EStop;  //Emergency Stop Pressed - VBL Rev0.1
      O     #FirstScanBit;  // Reset on first scan
      R     #UDTMotor.Command.ManRun;  // Reset Man Start command



NETWORK
TITLE = OUTPUT / Ausgabe
      A     #UDTMotor.Status.QOn;
      =     #q_On;



NETWORK
TITLE = FAILED TO RUN FAULT (FTR) / FEHLER BEIM AUSFÜHREN (FTR)
// Once the START_CMD output is issued from the PLC to the Motor/Pump, a 'Running' 
// feedback should be detected within a pre-set time. In the event of 
// non-receipt of the 'Running' feedback within this time, a Motor/Pump 'Fail to 
// Run' 
// alarm shall be generated.
// This alarm condition shall be maintained until the operator issues the 'Fault 
// Reset' command from the HMI. The Motor/Pump shall be made available for the 
// next operation, only after the 'Fault Reset'.
// 
// This alarm shall be generated only in the MCC-Auto Mode of operation.

// |************************************************************************|
// |                      Fail to Run fault Logic                           |
// |************************************************************************|

      A     #UDTMotor.Status.QOn;  // Motor/Pump Start command Present
      AN    #UDTMotor.Status.RunFb;  // Run Feedback Not Present
      AN    #UDTMotor.Command.AlarmMask;  // Fault are masked
      AN    #UDTMotor.Status.FTR;
      JC    FTRS;  // Yes!
      L     0;  // No! then initialise counter
      T     #UDTMotor.FTRActual;  // FTR_ACT (FTR) Timer-Counter
      JU    TMR1;

FTRS: A     #OneSec;  // 1 sec pulse
      JCN   TMR2;  // No!
      L     #UDTMotor.FTRActual;  // Increment @1sec
      L     1;
      +I;
      T     #UDTMotor.FTRActual;  // Update Timer-Counter

      T     #UDTMotor.ActiveTime;  // Time shown on HMI / SCADA

TMR2: L     #UDTMotor.FTRSet;  // FTR timer actual value
      L     #UDTMotor.FTRActual;  // FTR timer setpoint
      <=I;
      S     #UDTMotor.Status.FTR;  // Generate Motor/Pump Fail to Run Fault.(FTR)
TMR1: NOP   0;

NETWORK
TITLE = FAILED TO STOP FAULT (FTS)
// If the Motor/Pump START_CMD output from the PLC is de-energised due to any of 
// the 
// interlocks, then the running feedback should be lost within the preset time 
// . In the event of receipt of the running feedback even after this time, 
// a Motor/Pump 'Fail to Stop' alarm shall be generated.
// This alarm condition shall be maintained until the operator issues the 'Fault 
// Reset' command from the HMI. The Motor/Pump shall be made available for the 
// next operation only after the 'Fault Reset'.

// |************************************************************************|
// |                      Fail to Stop fault Logic                           |
// |************************************************************************|

      AN    #UDTMotor.Status.QOn;  // Motor/Pump Stop command Present
      A     #UDTMotor.Status.RunFb;  // Run Feedback Present
      AN    #UDTMotor.Command.AlarmMask;  // Fault are masked
      AN    #UDTMotor.Status.FTS;
      A     #UDTMotor.Command.FTSEn;  // FTS Enable
      JC    FTSS;  // Yes!
      L     0;  // No! then initialise counter
      T     #UDTMotor.FTSActual;  // FTS_ACT (FTS) Timer-Counter
      JU    TMR3;

FTSS: A     #OneSec;  // 1 sec pulse
      JCN   TMR4;  // No!
      L     #UDTMotor.FTSActual;  // Increment @1sec
      L     1;
      +I;
      T     #UDTMotor.FTSActual;  // Update Timer-Counter

      T     #UDTMotor.ActiveTime;  // Time shown on HMI / SCADA

TMR4: L     #UDTMotor.FTSSet;  // FTS timer actual value
      L     #UDTMotor.FTSActual;  // FTS timer setpoint
      <=I;
      S     #UDTMotor.Status.FTS;  // Generate Motor/Pump Fail to Stop Fault.(FTS)
TMR3: NOP   0;


NETWORK
TITLE = TRIPPED CONDITION LOGIC
// If the Motor/Pump loses process interlock in running mode or Tripped electrical 
// signal is lost, a Motor 'Tripped' alarm shall be generated.
// This alarm condition shall be maintained until the operator issues the 'Fault 
// Reset' command from the HMI. 
// 
// The Motor/Pump shall be made available for the next operation only after the 
// 'Fault 
// Reset'.

// |************************************************************************|
// |                                Tripped Logic                           |
// |************************************************************************|


      O(;
      A     #FeatureITripPolarity;  /// Feature bit=1.I_TrippedFB=1= Motor Tripped
      A     #i_TrippedFb;  // I_Tripped Signal 1 = Trip
      );

      O(;
      AN    #FeatureITripPolarity;  // Feature bit=0.I_TrippedFB=0= Motor Tripped
      AN    #i_TrippedFb;  // I_Tripped Signal 0 = Trip
      );

      O(;
      A     #UDTMotor.Status.QOn;  // Motor/Pump Start command Present
      AN    #UDTMotor.Status.Interlock;  // Process Interlock
      );
      S     #UDTMotor.Status.Tripped;




NETWORK
TITLE = DISCREPANCY LOGIC
// TIMER FOR DISCREPANCY LOGIC

// |************************************************************************|
// |                                    |
// |************************************************************************|

//      A     #UDTMotor.Command.DispcrEn// Motor/Pump Stop command Present
//      A     #UDTMotor.Command.AutoRun// Run Feedback Present
//      AN    #UDTMotor.Status.RunFb// Fault are masked
//      AN    #UDTMotor.Status.DiscrFault
// FTS Enable
//      JC    N1                   // Yes!
//      L     0                    // No! then initialise counter
//      T     #UDTMotor.PulseTimeStart// FTS_ACT (FTS) Timer-Counter
//      JU    N3

//N1:   A     #OneSec              // 1 sec pulse
//      JCN   N2                   // No!
//      L     #UDTMotor.PulseTimeStart// Increment @1sec
//      L     1
//      +I
//      T     #UDTMotor.PulseTimeStart// Update Timer-Counter

//N2:   NOP 0
//N3:   NOP 0


// |************************************************************************|
// |                   TIMER FOR DISCREPANCY LOGIC                 |
// |************************************************************************|

//      A     #UDTMotor.Command.DispcrEn// Motor/Pump Stop command Present
//      AN    #UDTMotor.Command.AutoRun// Run Feedback Present
//      A     #UDTMotor.Status.RunFb// Fault are masked
//      AN    #UDTMotor.Status.DiscrFault
// FTS Enable
//      JC    N11                  // Yes!
//      L     0                    // No! then initialise counter
//      T     #UDTMotor.PulseTimeStop// FTS_ACT (FTS) Timer-Counter
//      JU    N33

//N11:  A     #OneSec              // 1 sec pulse
//      JCN   N22                  // No!
//      L     #UDTMotor.PulseTimeStop// Increment @1sec
//      L     1
//      +I
//      T     #UDTMotor.PulseTimeStop// Update Timer-Counter

//N22:  NOP 0
//N33:  NOP 0



NETWORK
TITLE = DISCREPANCY LOGIC

//      A     #UDTMotor.Command.DispcrEn
//      A(                         // motor  Emergency stop not present
//      A     #UDTMotor.Command.AutoRun
//      A(
//      O     #UDTMotor.Status.FTR
//      O
//      AN    #UDTMotor.Status.RunFb
//      A(
//      L     #UDTMotor.PulseTimeStart
//      L     3
//      >I
//      )
//      )
//      O
//      AN    #UDTMotor.Command.AutoRun
//      A(
//      O     #UDTMotor.Status.FTS
//      O
//      A     #UDTMotor.Status.RunFb
//      A(
//      L     #UDTMotor.PulseTimeStop
//      L     3
//      >I
//      )
//      )
//      )
//      S     #UDTMotor.Status.DiscrFault

NETWORK
TITLE = FAULT RESET LOGIC
// Clear the faults on issue of Fault Reset command

// |************************************************************************|
// |                                   Fault Reset                          |
// |************************************************************************|

      A     #CommonReset;  // Commom fault command from HMI/SCADA
      FP    #UDTMotor.FP.CommonReset;
      S     #UDTMotor.Command.LocalFaultReset;  // Fault command from name plate

      O     #UDTMotor.Command.LocalFaultReset;  // Fault Reset Command from HMI
      O     #UDTMotor.Command.AlarmMask;  // Fault are masked
      R     #UDTMotor.Status.FTR;  // Motor/Pump Fail to Stop Fault.(FTS)
      R     #UDTMotor.Status.FTS;  // Motor/Pump tripped
      R     #UDTMotor.Status.Tripped;  // Clear the command
      R     #UDTMotor.Command.LocalFaultReset;
      R     #UDTMotor.Status.DiscrFault;

NETWORK
TITLE = GENERAL FAULT + ALARM LAMP + ALARM HOOTER
// ----------------------------------------------------------------------------------------------//
//                                GENERAL RESET                                                  //
// ----------------------------------------------------------------------------------------------//

// |************************************************************************|
// |                                  General Fault                         |
// |************************************************************************|

      O     #UDTMotor.Status.FTR;  // Motor/Pump Fail to Run Fault.(FTR)
      O     #UDTMotor.Status.FTS;  // Motor/Pump Fail to Stop Fault.(FTS)
      O     #UDTMotor.Status.Tripped;  // Motor/Pump tripped
      O     #UDTMotor.Status.DiscrFault;
      ON    #UDTMotor.Status.Inhibit;
      ON    #UDTMotor.Status.Remote;
      ON    #i_EStop;  // Emergency Stop
      =     #UDTMotor.Status.GeneralFault;  // Set the general Fault
      R     #UDTMotor.Command.ManRun;  // Motor/Pump Start - Stop command from HMI

//----------------------------------------------------------------------------------------------//
//                               ALARM LAMP                                                     //
//----------------------------------------------------------------------------------------------//
      A     #UDTMotor.Status.GeneralFault;
      S     #UDTMotor.Status.AlarmLampOut;

      AN    #UDTMotor.Status.GeneralFault;  // General fault
      FP    #UDTMotor.FP.GeneralFault;
      R     #UDTMotor.Status.AlarmLampOut;
//----------------------------------------------------------------------------------------------//
//                               ALARM HOOTER                                                   //
//----------------------------------------------------------------------------------------------//

      A     #UDTMotor.Status.GeneralFault;  // General fault
      FP    #UDTMotor.FP.Fault;
      S     #UDTMotor.Status.HooterOut;

      A     #HooterReset;
      R     #UDTMotor.Status.HooterOut;

NETWORK
TITLE = MOTOR /PUMP RUNNING HOUR LOGIC
// Run Hour Logic :
// The Motor/Pump running hours are updated based on the Motor/Pump running 
// feedback signal received from the MCC. These hours are calculated irrespective 
// of whether the Motor/Pump is in the Remote or Local Mode.

// **************************************************************************
// Start the CRH & ARH Second Counter for the preset value 3600.0
// **************************************************************************

      A     #UDTMotor.Status.RunFb;  // Motor/Pump Run Feedback Present
      A     #OneSec;  // 1 sec pulse
      JC    PRun;  // Yes! Then Goto 'Prun' label
      JU    Seg;  // No!  Then Goto 'Seg' label
PRun: L     #UDTMotor.TempARH;  // Current CRH Second Counter - Run Time Actual in Secs
      L     1;  // Increment @1sec
      +I;  // Add
      T     #UDTMotor.TempARH;  // Update CRH Second Counter- Run Time Actual in Secs

Seg:  NOP   0;



// |************************************************************************|
// |                      Actual Run Hour Logic                             |
// |************************************************************************|

// **************************************************************************
// Compare the Actual CRH Second Counter with the preset value 3600.0
// **************************************************************************

      A(;
      L     #UDTMotor.TempARH;  // Current CRH Second Counter- Run Time Actual in Secs
      L     3599;  // Load 3599 seconds
      >I;  // Current CRH counter greater then the 3599.0 seconds
      );
      JC    INC2;  // Yes ! Increment Cumulative Run Hours counter
      JU    SKP2;  // No!   Skip the logic for incrementing Cumulative Run Hours counter

// **************************************************************************
// Increment Actual Run Hour Counter
// **************************************************************************

INC2: L     #UDTMotor.ARH;  // Motor/Pump Cumulative Run timer actual value
      L     1;  // Load 1 Hour
      +I;  // Add the double word
      T     #UDTMotor.ARH;  // Transfer to Motor/Pump (CRH) Run HH Actual value

      L     0;  // Reset / Intialise
      T     #UDTMotor.TempARH;  // Current Second CRH Counter - Run Time Actual in Secs
SKP2: NOP   0;

// **************************************************************************
// Reset Actual Run Hour Counter
// **************************************************************************

      A     #UDTMotor.Command.ResetARH;
      O(;
      L     #UDTMotor.ARH;
      L     32000;
      >I;
      );
      JCN   SKP4;
      L     0;
      T     #UDTMotor.TempARH;
      T     #UDTMotor.ARH;
SKP4: R     #UDTMotor.Command.ResetARH;



NETWORK
TITLE = HMI ALARM BITS MAP

// HMI ALARM WORD MAP
      A     #UDTMotor.Status.FTR;
      =     #UDTMotor.AlarmHmi.%X8;

      A     #UDTMotor.Status.FTS;
      =     #UDTMotor.AlarmHmi.%X9;

      A     #UDTMotor.Status.Tripped;
      =     #UDTMotor.AlarmHmi.%X10;

      A     #UDTMotor.Status.FTRReverse;
      =     #UDTMotor.AlarmHmi.%X11;

      A     #UDTMotor.Status.GeneralFault;
      =     #UDTMotor.AlarmHmi.%X12;

      A     #UDTMotor.Status.InlkBypassIcon;
      =     #UDTMotor.AlarmHmi.%X13;

      A     #UDTMotor.Status.InlkStatusIcon;
      =     #UDTMotor.AlarmHmi.%X14;

      A     #UDTMotor.Status.RunFb;
      =     #UDTMotor.AlarmHmi.%X15;

      A     #UDTMotor.Status.Spare1;
      =     #UDTMotor.AlarmHmi.%X0;

      A     #UDTMotor.Status.Mode;
      =     #UDTMotor.AlarmHmi.%X1;

      A     #UDTMotor.Status.AlarmMask;
      =     #UDTMotor.AlarmHmi.%X2;

      A     #UDTMotor.Status.SimOn;
      =     #UDTMotor.AlarmHmi.%X3;

      AN    #UDTMotor.Status.Remote;
      =     #UDTMotor.AlarmHmi.%X4;

      AN    #UDTMotor.Status.Inhibit;
      =     #UDTMotor.AlarmHmi.%X5;




NETWORK
TITLE = MOTOR/PUMP HMI DISPLAY ON HMI FTR/FTS, TRIPPED, RUNing, STOPPED
// 0 - STOPPED
// 1 - RUNNING
// 2 - TRIPPED
// 3 - FTR / FTS
// **************************************************************************
// FAULT INDICATION ON HMI
// **************************************************************************


      O     #UDTMotor.Status.FTR;  // Motor/Pump Fail to Run Fault.(FTR)
      O     #UDTMotor.Status.FTS;  // Motor/Pump Fail to Run Fault.(FTS)
      JCN   F1;
      L     3;
      JU    F6;


// **************************************************************************
// TRIPPED INDICATION ON HMI
// **************************************************************************


F1:   O     #UDTMotor.Status.Tripped;
      JCN   F2;
      L     2;
      JU    F6;


// **************************************************************************
// RUNNING INDICATION ON HMI
// **************************************************************************

F2:   A     #UDTMotor.Status.QOn;  // Motor/Pump Running remote
      A     #UDTMotor.Status.RunFb;
      JCN   F3;
      L     1;
      JU    F6;

// **************************************************************************
//  STARTING INDICATION ON HMI
// **************************************************************************

F3:   A     #UDTMotor.Status.QOn;  // Motor/Pump Without RunFeedback remote
      AN    #UDTMotor.Status.RunFb;
      JCN   F4;
      L     4;
      JU    F6;


// **************************************************************************
//  STOPING INDICATION ON HMI
// **************************************************************************

F4:   AN    #UDTMotor.Status.QOn;  // Motor/Pump Without RunFeedback remote
      A     #UDTMotor.Status.RunFb;  // Motor Feedback
      AN    #UDTMotor.Status.FTS;  // Fail To Stop
      JCN   F5;
      L     5;
      JU    F6;


// STOPPED INDICATION ON HMI
// **************************************************************************
F5:   L     0;

// **************************************************************************
// DISPLAY INDICATION ON HMI
// **************************************************************************

F6:   T     #UDTMotor.Display;


NETWORK
TITLE = CM Revision Details
// |************************************************************************|
// |                       CM Revision Number                               |
// |************************************************************************|
      L     3.5;  //Revision Number
      T     #UDTMotor.PLCVersionNo;  //Current Version number of the Library

NETWORK
TITLE = SAVE TEMP DATA TO DB
      OPN   DB [#DB];

      L     %LW0;  // Data transfer back to DB Area
      T     W [AR1, P#0.0];

      L     %LW2;  // Data transfer back to DB Area
      T     W [AR1, P#2.0];

      L     %LW4;  // Data transfer back to DB Area
      T     W [AR1, P#4.0];

      L     %LW6;  // Data transfer back to DB Area
      T     W [AR1, P#6.0];


      L     #UDTMotor.FTRSet;  // Data transfer back to DB Area
      T     W [AR1, P#8.0];

      L     #UDTMotor.FTSSet;  // Data transfer back to DB Area
      T     W [AR1, P#10.0];

      L     #UDTMotor.FTRActual;  // Data transfer back to DB Area
      T     W [AR1, P#12.0];

      L     #UDTMotor.FTSActual;  // Data transfer back to DB Area
      T     W [AR1, P#14.0];

      L     #UDTMotor.ARH;  // Data transfer back to DB Area
      T     W [AR1, P#16.0];

      L     #UDTMotor.Display;  // Data transfer back to DB Area
      T     W [AR1, P#18.0];

      L     #UDTMotor.TempARH;  // Data transfer back to DB Area
      T     W [AR1, P#20.0];

      L     #UDTMotor.PulseTimeStart;
      T     W [AR1, P#22.0];  // Data transfer to Local Area

      L     #UDTMotor.PulseTimeStop;
      T     W [AR1, P#24.0];  // Data transfer to Local Area

      L     #UDTMotor.BypassPermissive;
      T     W [AR1, P#26.0];  // Data transfer to Local Area

      L     #UDTMotor.BypassInterlock;
      T     W [AR1, P#28.0];  // Data transfer to Local Area

      L     %LW30;
      T     W [AR1, P#30.0];  // Data transfer to Local Area

      L     %LW32;
      T     W [AR1, P#32.0];  // Data transfer to Local Area

      L     #UDTMotor.AlarmHmi;
      T     W [AR1, P#34.0];  // Data transfer to Local Area

      L     #UDTMotor.ActiveTime;
      T     W [AR1, P#36.0];  // Data transfer to Local Area

      L     #UDTMotor.MotorType;
      T     W [AR1, P#38.0];  // Data transfer to Local Area

      L     #UDTMotor.Spare2;
      T     D [AR1, P#40.0];  // Data transfer to Local Area

      L     %LD44;
      T     D [AR1, P#44.0];  // Data transfer to Local Area

      L     %LW48;
      T     W [AR1, P#48.0];  // Data transfer to Local Area

//Load Library Version number to display on UI
      L     #UDTMotor.PLCVersionNo;  //Current Version number of the Library
      T     D [AR1, P#50.0];

END_FUNCTION
